// TIA Portal V21 export
VAR_GLOBAL   // PLC tag table "Inputs"
   DI_EmergencyStop AT %I0.0 : Bool;   //    {ExternalWritable false}
   DI_Reset AT %I0.1 : Bool;   //    {ExternalWritable false}
   DI_ContactorON_Pump1 AT %I0.4 : Bool;   //    {ExternalWritable false}
   DI_SoftstartON_Pump1 AT %I0.5 : Bool;   //    {ExternalWritable false}
   DI_SoftstartBypassed_Pump1 AT %I0.6 : Bool;   //    {ExternalWritable false}
   DI_SoftstartFault_Pump1 AT %I0.7 : Bool;   //    {ExternalWritable false}
   DI_Protection_Pump1 AT %I1.0 : Bool;   //    {ExternalWritable false}
   DI_ContactorON_Pump2 AT %I1.1 : Bool;   //    {ExternalWritable false}
   DI_SoftstartON_Pump2 AT %I1.2 : Bool;   //    {ExternalWritable false}
   DI_SoftstartBypassed_Pump2 AT %I1.3 : Bool;   //    {ExternalWritable false}
   DI_SoftstartFault_Pump2 AT %I1.4 : Bool;   //    {ExternalWritable false}
   DI_Protection_Pump2 AT %I1.5 : Bool;   //    {ExternalWritable false}
   AI_TankLevel1 AT %IW10 : Int;   //    {ExternalWritable false}
   AI_TankLevel2 AT %IW12 : Int;   //    {ExternalWritable false}
   DI_Start AT %I0.2 : Bool;   //    {ExternalWritable false}
   DI_Stop AT %I0.3 : Bool;   //    {ExternalWritable false}
   DI_Reserve_1_6 AT %I1.6 : Bool;   //    {ExternalWritable false}
   DI_Reserve_1_7 AT %I1.7 : Bool;   //    {ExternalWritable false}
END_VAR
